FUNCTION_BLOCK AXIS
VAR_INPUT	
	tAmsNetId: T_AmsNetId := '192.168.0.33.1.1';  	
	tAmsPort: T_AmsPort := 501;
	
	rVel: REAL := 75.0;
	rAcc: REAL := 3000.0;
	rDec: REAL := 3000.0;
	rJerk: REAL := 72000.0;
	
	mcrs: MC_ReadStatus := (Enable:=TRUE);
	mcrae: MC_ReadAxisError := (Enable:=TRUE);
	mcp: MC_Power := (Enable:=FALSE, Enable_Positive:=TRUE, Enable_Negative:=TRUE);
	mcr: MC_Reset;
	mcs: MC_Stop;
	mch: MC_Home;
	mcma: MC_MoveAbsolute;
	mcmr: MC_MoveRelative;
	mcmv: MC_MoveVelocity := (Direction := -1);// 1 Positiv, -1 Negativ
	rOffsetHoming: REAL  := -45.0;
END_VAR
VAR_OUTPUT	
	bError: BOOL;
	iStep: INT;
	rActPos: REAL;
	rActVel: REAL;
	rActAcc: REAL;
END_VAR
VAR_IN_OUT
	axis: AXIS_REF;
END_VAR
VAR
	dVel: LREAL;
	dAcc: LREAL;
	dDec: LREAL;	
	dJerk: LREAL;

	dActPos: LREAL;
	dActVel: LREAL;
	dActAcc: LREAL;	
	
	rExtVel: REAL;
	rExtAcc: REAL;

	dExtVel: LREAL;
	dExtAcc: LREAL;
	dExtPos: LREAL;
	diExtDir: DINT;
	
	// Regler für die Ansteuerung der Achsen
	// Position/Winkel

	// Geschwindigkeit/Winkeländerung
	bCtrlEnable_v_RST: BOOL := TRUE;
	
	
	rE_ExtPos: REAL;
	rE_ExtVel: REAL;
		
	adsread_kv: ADSREAD;
	adswrite_kv: ADSWRITE;
	dKvRead: LREAL;
	dKvWrite: LREAL;
	iStepAds: INT;
	
	bDummy: BOOL;
	rDummy: REAL;
	dDummy: LREAL;
	
END_VAR

// Aufruf der PLC OPEN Motionbausteine
dVel := REAL_TO_LREAL(rVel);
dAcc := REAL_TO_LREAL(rAcc);
dDec := REAL_TO_LREAL(rDec);
dJerk := REAL_TO_LREAL(rJerk);
PLC_OPEN();

bError := mch.Error OR mcs.Error OR mcmr.Error OR mcma.Error OR mcmv.Error;

// Zuweisung der Motion Control Istwerte
dActPos := axis.NcToPlc.ActPos;
dActVel := axis.NcToPlc.ActVelo;
dActAcc := axis.NcToPlc.ActAcc;
rActPos := LREAL_TO_REAL(dActPos);
rActVel := LREAL_TO_REAL(dActVel);
rActAcc := LREAL_TO_REAL(dActAcc);

ACTION EXECUTE_TO_FALSE:
mcr.Execute := FALSE;
mcs.Execute := FALSE;
mch.Execute := FALSE;
mcma.Execute := FALSE;
mcmr.Execute := FALSE;
mcmv.Execute := FALSE;
END_ACTION

ACTION PLC_OPEN:
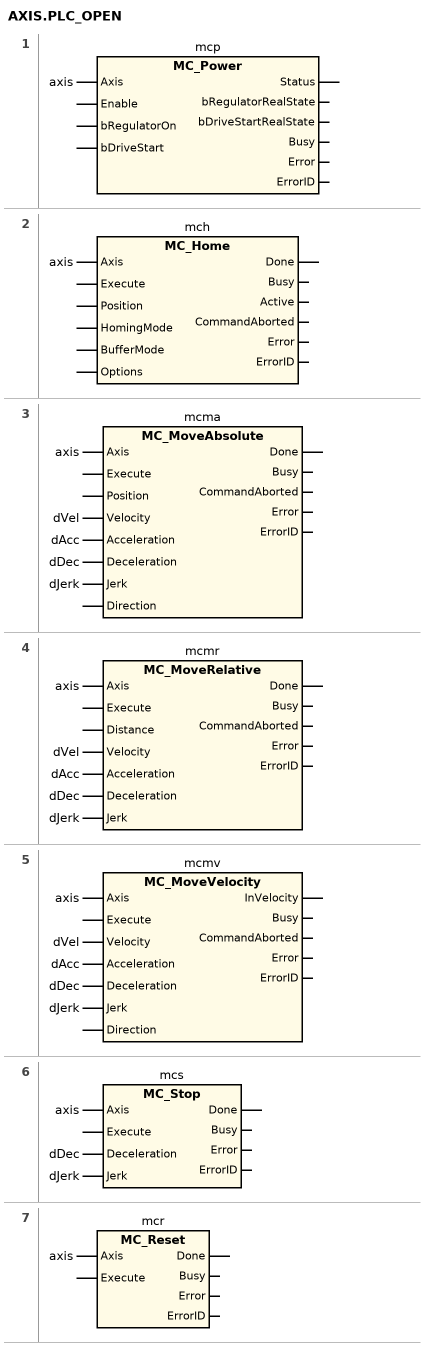
// NETWORK 1
mcp(Axis := axis); // MC_Power

// NETWORK 2
mch(Axis := axis); // MC_Home

// NETWORK 3
mcma(Axis := axis, Velocity := dVel, Acceleration := dAcc, Deceleration := dDec, Jerk := dJerk); // MC_MoveAbsolute

// NETWORK 4
mcmr(Axis := axis, Velocity := dVel, Acceleration := dAcc, Deceleration := dDec, Jerk := dJerk); // MC_MoveRelative

// NETWORK 5
mcmv(Axis := axis, Velocity := dVel, Acceleration := dAcc, Deceleration := dDec, Jerk := dJerk); // MC_MoveVelocity

// NETWORK 6
mcs(Axis := axis, Deceleration := dDec, Jerk := dJerk); // MC_Stop

// NETWORK 7
mcr(Axis := axis); // MC_Reset

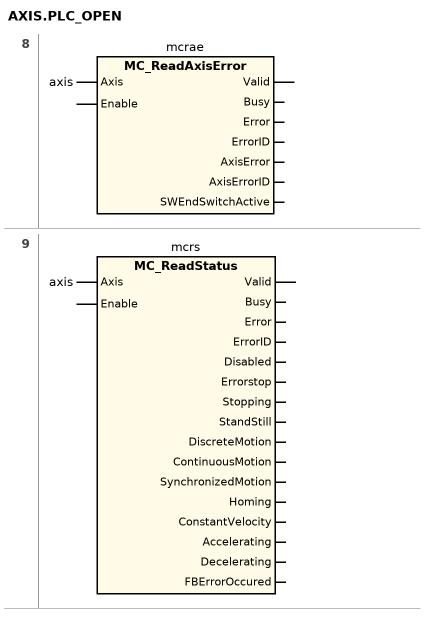
// NETWORK 8
mcrae(Axis := axis); // MC_ReadAxisError

// NETWORK 9
mcrs(Axis := axis); // MC_ReadStatus
END_ACTION

END_FUNCTION_BLOCK

(* stored: Version 1.1.0.1, ProductVersion 3.1.4024.10
   POU AXIS: Id {390966a0-822b-40fb-8d29-74dcb1896894}, SpecialFunc None
   Action EXECUTE_TO_FALSE: Id {72290231-c133-4610-97eb-5daf65cfd1a7}
   Action PLC_OPEN: Id {b5925376-31a1-4115-99f8-55ecedd36e40} *)
